Omron CX-Programmer project NewProject (CX-Programmer 9.73)

# PLC NewPLC1: CP1E N60

## Global symbols (name address type ; comment)
0.00 BOOL  ; BUTTONS YELLOW
100.00 BOOL  ; RED
100.01 BOOL  ; YELLOW
100.02 BOOL  ; GREEN
10.00 BOOL  ; BUTTONSRED
T000 BOOL  ; BUTTONS YELLOW
T001 BOOL  ; STOP
T002 BOOL  ; STOP GREEN
M1 BOOL

## Program NewProgram1 (cyclic task 0)
Local symbols
Y1 BOOL

### Section Section1

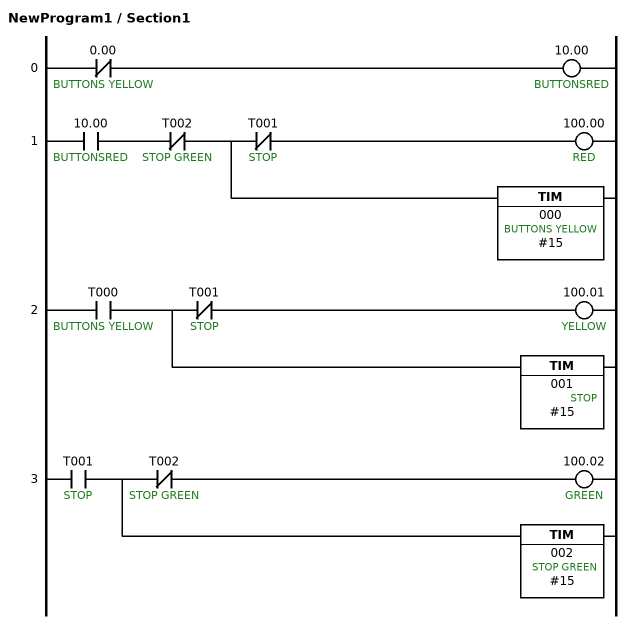
; rung 0
LDNOT 0.00  ; BUTTONS YELLOW
OUT 10.00  ; BUTTONSRED
; rung 1
LD 10.00  ; BUTTONSRED
ANDNOT T002  ; STOP GREEN
OUT TR0
ANDNOT T001  ; STOP
OUT 100.00  ; RED
LD TR0
TIM 000 #15  ; BUTTONS YELLOW
; rung 2
LD T000  ; BUTTONS YELLOW
OUT TR0
ANDNOT T001  ; STOP
OUT 100.01  ; YELLOW
LD TR0
TIM 001 #15  ; STOP
; rung 3
LD T001  ; STOP
OUT TR0
ANDNOT T002  ; STOP GREEN
OUT 100.02  ; GREEN
LD TR0
TIM 002 #15  ; STOP GREEN

### Section END
; rung 0
END(001)